TYPE ServicesTimingStatuses :
STRUCT
	healthStatus: HealthStatus;
	busyStatus: BusyStatus;
END_STRUCT
END_TYPE

(* stored: Version 1.1.0.1, ProductVersion 3.1.4019.2
   DUT ServicesTimingStatuses: Id {3a2f0421-9975-4b6c-85b1-a10d930095ce} *)
